FUNCTION_BLOCK FB_Basis_Objekt_Sensor
VAR_INPUT
END_VAR
VAR_OUTPUT
END_VAR
VAR
END_VAR

END_FUNCTION_BLOCK

(* stored: Version 1.1.0.1
   POU FB_Basis_Objekt_Sensor: Id {6644944f-8e65-458a-9a73-3fb96675b87b}, SpecialFunc None *)
